FUNCTION F_Random : LREAL
VAR_INPUT
END_VAR
VAR
	nSeed 		: INT;
	rand		: DRAND;
	fbCpu		: GETCPUCOUNTER;
	nLow		: DWORD;
END_VAR

fbCpu(cpuCntLoDW => nLow);
nSeed := TO_INT(nLow);
rand(Seed:=nSeed);
F_Random := rand.Num;

END_FUNCTION

(* stored: Version 1.1.0.1, ProductVersion 3.1.4026.18
   POU F_Random: Id {7bd08c84-9c8b-465f-8e53-5e71d356327c}, SpecialFunc None *)
